// TIA Portal V20 export
// export: Created 2026-08-08T00:00:00.0000000Z, ExportSetting WithDefaults, DisplayName Totally Integrated Automation Portal, DisplayVersion V20, DisplayName TIA Portal Openness, DisplayVersion V20, DisplayName TIA Portal Version Control Interface, DisplayVersion V20, DisplayName STEP 7 Professional, DisplayVersion V20, DisplayName STEP 7 Safety, DisplayVersion V20, DisplayName WinCC Basic/Comfort/Advanced, DisplayVersion V20, DisplayName WinCC Professional, DisplayVersion V20, DisplayName WinCC Unified, DisplayVersion V20
DATA_BLOCK "IO_Buffer_DB"   // DB
{ S7_Optimized_Access := 'TRUE' }
VERSION : 0.1
// Abstract channel table: DI[1..368] covers all 23 DI16 modules across AFT/MID/FWD (7+7+9), DQ[1..208] covers all 13 DQ16 modules (4+4+5) - matches the confirmed BOM module counts. Index N here is OUR OWN channel numbering, not a real %I/%Q address - FC_IoMapper is the only place real physical addresses get referenced, once the hardware address assignment question (see FC_IoMapper header comment) is resolved.
// stored: AutoNumber true, IsOnlyStoredInLoadMemory false, IsRetainMemResEnabled false, IsWriteProtectedInAS false, MemoryReserve 100
   VAR
      DI : Array[1..368] of Bool;
      DQ : Array[1..208] of Bool;
   END_VAR
BEGIN
END_DATA_BLOCK
